# EPICS substitutions: iocBoot/iocHindsXray/asynRecord.substitutions
file "$(ASYN)/db/asynRecord.db"
{
pattern
{P              R         PORT     ADDR  OMAX IMAX}
{HindsXray:    serial1   serial1    0    256  256}
{HindsXray:    serial2   serial2    0    256  256}
{HindsXray:    serial3   serial3    0    256  256}
{HindsXray:    serial8   PMAC_IP    0    256  256}
}
